{attribute 'qualified_only'}
TYPE E_SerialState :
(
	eStopped := 0,
	eSearchForHeader,
	eReceive
);
END_TYPE

(* stored: Version 1.1.0.1, ProductVersion 3.1.4024.9
   DUT E_SerialState: Id {968294fa-a157-4444-be83-0f0cf76275fc} *)
